FUNCTION_BLOCK TimeOptimalTrajectory
VAR_INPUT
	currentPose			: RobotPoseSimple;
	drive				: BOOL 				:= FALSE;
END_VAR
VAR_OUTPUT
	finished			: BOOL 				:= FALSE;
	ready				: BOOL				:= FALSE;
	generationFailed	: BOOL				:= FALSE;
	pathReady			: BOOL				:= FALSE;
	referencePose		: RobotPoseSimple;
	referenceVelocities	: RobotPoseSimple;
	WPLidx 				: INT 				:= 0;
	path				: Path;
END_VAR
VAR
	trajectoryPlanner	: TrajectoryPlanner;
	wayPointListRaw		: ARRAY [0..100] OF RobotPoseSimple;
	cnt					: INT 				:= 0;
	
    maxRadius		    : LREAL				:= ControlParameters.maxRadius;
	
	samplingTime		: LREAL				:= ControlParameters.samplingTime;
	
	maxVel				: LREAL				:= ControlParameters.maxVel;
	maxAcc				: LREAL				:= ControlParameters.maxAcc;
	
	arcLengthSlow		: LREAL				:= ControlParameters.arcLengthSlow;
	maxSlowVel			: LREAL				:= ControlParameters.maxSlowVel;
	
	maxRotVel			: LREAL				:= ControlParameters.maxRotVel;
	maxRotAcc			: LREAL				:= ControlParameters.maxRotAcc;
	
	thetaDZ				: LREAL				:= ControlParameters.thetaDZ;
	
END_VAR

ready 				:= trajectoryPlanner.trajectoriesReady;
generationFailed	:= trajectoryPlanner.trajectoryGenerationFailed;
pathReady 			:= path.ready;

IF cnt = LREAL_TO_INT(samplingTime/Var_HAWIno.CONTROLLER_CYCLE_TIME) AND NOT finished THEN
	WPLidx := WPLidx +1;
	cnt := 0;
END_IF

IF  trajectoryPlanner.posTrajectory[WPLidx].x = -1 AND trajectoryPlanner.posTrajectory[WPLidx].y = -1  AND trajectoryPlanner.posTrajectory[WPLidx].theta = -1 THEN
	finished := TRUE;
END_IF

IF drive AND NOT finished AND ready THEN
	referencePose := trajectoryPlanner.posTrajectory[WPLidx];
	referenceVelocities := trajectoryPlanner.velTrajectory[WPLidx];
	cnt := cnt +1;	
END_IF

METHOD generateTrajectory : BOOL
VAR_INPUT
END_VAR
trajectoryPlanner.generateTrajectory();
END_METHOD

METHOD reset : BOOL
VAR_INPUT
END_VAR
WPLidx 			:= 0; 						//reset
finished 		:= FALSE;

path.reset();
trajectoryPlanner.reset();
reset := TRUE;
END_METHOD

METHOD setRobotPose : RobotPoseSimple
VAR_INPUT
	newPose: RobotPoseSimple;
END_VAR
//not needed here
END_METHOD

METHOD setWaypointList : ARRAY [0..100] OF RobotPoseSimple
VAR_INPUT
	newWayPointList	: ARRAY [0..100]  OF RobotPoseSimple;
END_VAR

VAR
	extendedWayPointList			:	ARRAY [0..101] OF RobotPoseSimple;
	i								: INT;
	maxInitialPoseError				: LREAL := 35;		// unit: mm
END_VAR
// Insert actual position as first waypoint if robot is too far away from first
IF (SQRT(EXPT(currentPose.x - newWayPointList[0].x, 2) + EXPT(currentPose.y - newWayPointList[0].y, 2)) > maxInitialPoseError) AND currentPose.x <> 0 AND currentPose.y <> 0 THEN
	// shift all elements +1 to right except the lat one (gets overwritten)
	FOR i := 100 TO 0 BY -1 DO
		extendedWayPointList[i + 1] := newWayPointList[i];
	END_FOR

	// insert actual pose as first waypoint
	extendedWayPointList[0] := currentPose;
ELSE
	// shift all elements +1 to right except the lat one (gets overwritten)
	FOR i := 0 TO 100 BY 1 DO
		extendedWayPointList[i] := newWayPointList[i];
	END_FOR
	
	extendedWayPointList[101].x := -1;
	extendedWayPointList[101].y := -1;
	extendedWayPointList[0].theta := currentPose.theta;
END_IF

path(waypointListRaw := extendedWayPointList, maxRadius := maxRadius, thetaDZ := thetaDZ);

IF path.ready THEN
	trajectoryPlanner(path := path, 
				  qAccMax := maxAcc, 
				  qVelMax := maxVel, 
				  thetaAccMax := maxRotAcc,
				  thetaVelMax := maxRotVel,
				  qVelMaxSlow := maxSlowVel,
				  arcLengthSlow := arcLengthSlow,
				  deltaT := samplingTime);
 END_IF
END_METHOD

END_FUNCTION_BLOCK

(* stored: Version 1.1.0.1, ProductVersion 3.1.4024.11
   POU TimeOptimalTrajectory: Id {c9d800de-1da9-4b82-a21b-c146282eb721}, SpecialFunc None
   Method generateTrajectory: Id {3d1dbbe1-33ce-40a6-ae71-929ba959894c}
   Method reset: Id {a510e6d9-b061-4cba-a683-d76415bcb2be}
   Method setRobotPose: Id {612c742a-1fe7-4003-9836-d6bbc0467a35}
   Method setWaypointList: Id {e85e045f-80a3-4da6-9e39-79af30febaa9} *)
